// TIA Portal V17 export
// export: Created 2022-06-27T14:00:24.4169132Z, ExportSetting WithDefaults, DisplayName Totally Integrated Automation Portal, DisplayVersion V17 Update 3, DisplayName TIA Portal Openness, DisplayVersion V17 Update 3, DisplayName TIA Portal Version Control Interface, DisplayVersion V17, DisplayName SINAMICS Startdrive Advanced, DisplayVersion V17 Update1, DisplayName SINAMICS Startdrive G110M, G120, G120C, G120D, G120P, G115D, DisplayVersion V17 Update1, DisplayName SINAMICS Startdrive G130, G150, S120, S150, SINAMICS MV, S210, DisplayVersion V17 Update1, DisplayName STEP 7 Professional, DisplayVersion V17 Update 3, DisplayName STEP 7 Safety, DisplayVersion V17, DisplayName WinCC UA Professional, DisplayVersion V17 Update 3
FUNCTION_BLOCK "S0832_TRENDS_CONTROL"   // FB832, LAD
{ S7_Optimized_Access := 'TRUE' }
VERSION : 0.1
// stored: AutoNumber false, IsIECCheckEnabled false, IsRetainMemResEnabled false, MemoryReserve 100, SetENOAutomatically false, UDAEnableTagReadback false
   VAR
      ls_iIteration1 : Int;
      ls_stcConfigTrendEditC1Dry { S7_SetPoint := 'True'} : "S0831_TREND_CONFIG";
      ls_stcConfigTrendEditC1Roast { S7_SetPoint := 'True'} : "S0831_TREND_CONFIG";
      ls_stcConfigTrendEditC2Dry { S7_SetPoint := 'True'} : "S0831_TREND_CONFIG";
      ls_stcConfigTrendEditC2Roast { S7_SetPoint := 'True'} : "S0831_TREND_CONFIG";
      ls_stcConfigTrendVisuC1Dry { S7_SetPoint := 'True'} : "S0831_TREND_CONFIG";
      ls_stcConfigTrendVisuC1Roast { S7_SetPoint := 'True'} : "S0831_TREND_CONFIG";
      ls_stcConfigTrendVisuC2Dry { S7_SetPoint := 'True'} : "S0831_TREND_CONFIG";
      ls_stcConfigTrendVisuC2Roast { S7_SetPoint := 'True'} : "S0831_TREND_CONFIG";
   END_VAR
   VAR_TEMP   // added for the SCL form of the ladder/FBD networks
      _w1 : Bool;
   END_VAR
BEGIN

REGION Network 1 (SCL): SCL transferencia de valores da receita em edicao para o bloco de trend / Move valores edicao camara 1
   REGION Move valores das receitas em edicao para o bloco de trend
       REGION Move valores do secador para o bloco de trend
           FOR #ls_iIteration1 := 1 TO 10 DO
               // Statement section FOR
               #ls_stcConfigTrendEditC1Dry.i_arXBottom[#ls_iIteration1] := "S0921_ManipulacaoReceitas_DB".RecipeEdit.C1ProfileDry.arCoffeeTemperature[#ls_iIteration1];
               #ls_stcConfigTrendEditC1Dry.i_arYLeft[#ls_iIteration1] := "S0921_ManipulacaoReceitas_DB".RecipeEdit.C1ProfileDry.arInletTemperature[#ls_iIteration1];
               #ls_stcConfigTrendEditC1Dry.i_arYRight[#ls_iIteration1] := "S0921_ManipulacaoReceitas_DB".RecipeEdit.C1ProfileDry.arBlowerSpeed[#ls_iIteration1];
           END_FOR;
           #ls_stcConfigTrendEditC1Dry.i_rCorte := "S0921_ManipulacaoReceitas_DB".RecipeEdit.Recipe.rC1DryTemperature;
           #ls_stcConfigTrendEditC1Dry.i_rAromatizacao := 0.0;
       END_REGION
       REGION Move valores do torrador para o bloco de trend
           FOR #ls_iIteration1 := 1 TO 10 DO
               // Statement section FOR
               #ls_stcConfigTrendEditC1Roast.i_arXBottom[#ls_iIteration1] := "S0921_ManipulacaoReceitas_DB".RecipeEdit.C1ProfileRoast.arCoffeeTemperature[#ls_iIteration1];
               #ls_stcConfigTrendEditC1Roast.i_arYLeft[#ls_iIteration1] := "S0921_ManipulacaoReceitas_DB".RecipeEdit.C1ProfileRoast.arInletTemperature[#ls_iIteration1];
               #ls_stcConfigTrendEditC1Roast.i_arYRight[#ls_iIteration1] := "S0921_ManipulacaoReceitas_DB".RecipeEdit.C1ProfileRoast.arBlowerSpeed[#ls_iIteration1];
           END_FOR;
           #ls_stcConfigTrendEditC1Roast.i_rCorte := "S0921_ManipulacaoReceitas_DB".RecipeEdit.Recipe.rC1RoastCutTemperature;
           #ls_stcConfigTrendEditC1Roast.i_rAromatizacao := "S0921_ManipulacaoReceitas_DB".RecipeEdit.Recipe.rC1RoastQuenchTemperature;
       END_REGION
   END_REGION
END_REGION

REGION Network 2: Bloco de trend da edicao de receita / Chama blocos edicao camara 1
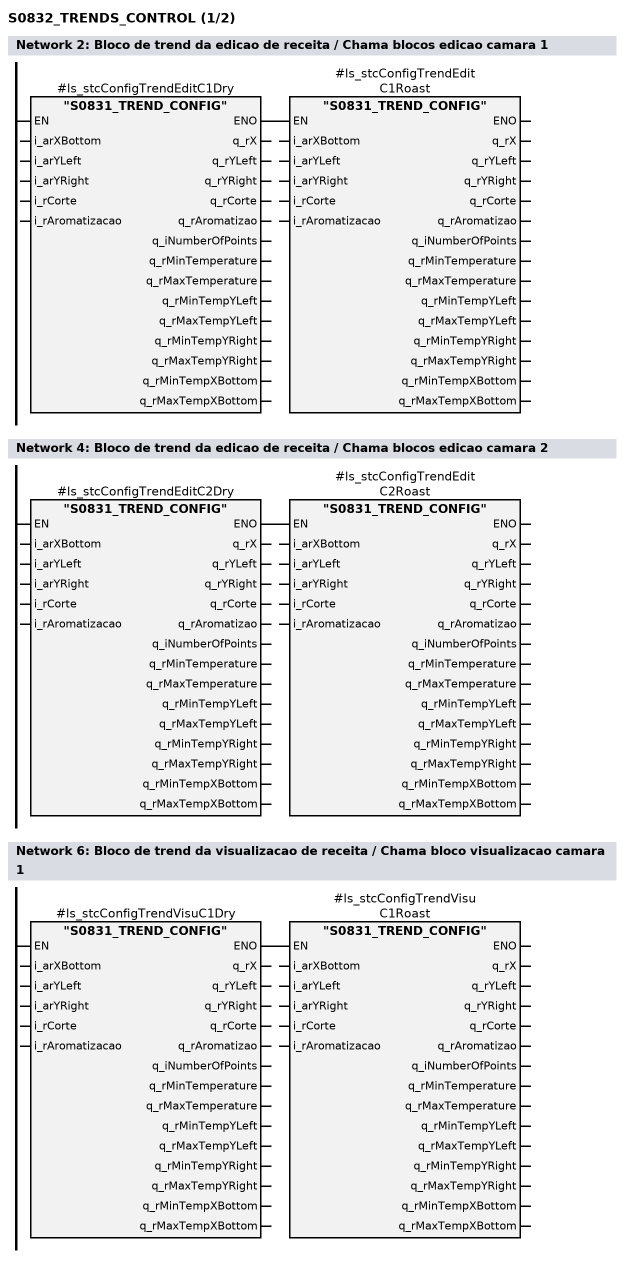
   RUNG wire#powerrail
      #ls_stcConfigTrendEditC1Dry(i_arXBottom :=, i_arYLeft :=, i_arYRight :=, i_rCorte :=, i_rAromatizacao :=, q_rX =>, q_rYLeft =>, q_rYRight =>, q_rCorte =>, q_rAromatizao =>, q_iNumberOfPoints =>, q_rMinTemperature =>, q_rMaxTemperature =>, q_rMinTempYLeft =>, q_rMaxTempYLeft =>, q_rMinTempYRight =>, q_rMaxTempYRight =>, q_rMinTempXBottom =>, q_rMaxTempXBottom =>)
      #ls_stcConfigTrendEditC1Roast(i_arXBottom :=, i_arYLeft :=, i_arYRight :=, i_rCorte :=, i_rAromatizacao :=, q_rX =>, q_rYLeft =>, q_rYRight =>, q_rCorte =>, q_rAromatizao =>, q_iNumberOfPoints =>, q_rMinTemperature =>, q_rMaxTemperature =>, q_rMinTempYLeft =>, q_rMaxTempYLeft =>, q_rMinTempYRight =>, q_rMaxTempYRight =>, q_rMinTempXBottom =>, q_rMaxTempXBottom =>)
   END_RUNG
   // the same network as SCL:
   #ls_stcConfigTrendEditC1Dry(ENO => #_w1);   // "S0831_TREND_CONFIG"
   IF #_w1 THEN
       #ls_stcConfigTrendEditC1Roast();   // "S0831_TREND_CONFIG"
   END_IF;
END_REGION

REGION Network 3 (SCL): SCL transferencia de valores da receita em edicao para o bloco de trend / Move valores edicao camara 2
   REGION Move valores das receitas em edicao para o bloco de trend
       REGION Move valores do secador para o bloco de trend
           FOR #ls_iIteration1 := 1 TO 10 DO
               // Statement section FOR
               #ls_stcConfigTrendEditC2Dry.i_arXBottom[#ls_iIteration1] := "S0921_ManipulacaoReceitas_DB".RecipeEdit.C2ProfileDry.arCoffeeTemperature[#ls_iIteration1];
               #ls_stcConfigTrendEditC2Dry.i_arYLeft[#ls_iIteration1] := "S0921_ManipulacaoReceitas_DB".RecipeEdit.C2ProfileDry.arInletTemperature[#ls_iIteration1];
               #ls_stcConfigTrendEditC2Dry.i_arYRight[#ls_iIteration1] := "S0921_ManipulacaoReceitas_DB".RecipeEdit.C2ProfileDry.arBlowerSpeed[#ls_iIteration1];
           END_FOR;
           #ls_stcConfigTrendEditC2Dry.i_rCorte := "S0921_ManipulacaoReceitas_DB".RecipeEdit.Recipe.rC2DryTemperature;
           #ls_stcConfigTrendEditC2Dry.i_rAromatizacao := 0.0;
       END_REGION
       REGION Move valores do torrador para o bloco de trend
           FOR #ls_iIteration1 := 1 TO 10 DO
               // Statement section FOR
               #ls_stcConfigTrendEditC2Roast.i_arXBottom[#ls_iIteration1] := "S0921_ManipulacaoReceitas_DB".RecipeEdit.C2ProfileRoast.arCoffeeTemperature[#ls_iIteration1];
               #ls_stcConfigTrendEditC2Roast.i_arYLeft[#ls_iIteration1] := "S0921_ManipulacaoReceitas_DB".RecipeEdit.C2ProfileRoast.arInletTemperature[#ls_iIteration1];
               #ls_stcConfigTrendEditC2Roast.i_arYRight[#ls_iIteration1] := "S0921_ManipulacaoReceitas_DB".RecipeEdit.C2ProfileRoast.arBlowerSpeed[#ls_iIteration1];
           END_FOR;
           #ls_stcConfigTrendEditC2Roast.i_rCorte := "S0921_ManipulacaoReceitas_DB".RecipeEdit.Recipe.rC2RoastCutTemperature;
           #ls_stcConfigTrendEditC2Roast.i_rAromatizacao := "S0921_ManipulacaoReceitas_DB".RecipeEdit.Recipe.rC2RoastQuenchTemperature;
       END_REGION
   END_REGION
END_REGION

REGION Network 4: Bloco de trend da edicao de receita / Chama blocos edicao camara 2
   RUNG wire#powerrail
      #ls_stcConfigTrendEditC2Dry(i_arXBottom :=, i_arYLeft :=, i_arYRight :=, i_rCorte :=, i_rAromatizacao :=, q_rX =>, q_rYLeft =>, q_rYRight =>, q_rCorte =>, q_rAromatizao =>, q_iNumberOfPoints =>, q_rMinTemperature =>, q_rMaxTemperature =>, q_rMinTempYLeft =>, q_rMaxTempYLeft =>, q_rMinTempYRight =>, q_rMaxTempYRight =>, q_rMinTempXBottom =>, q_rMaxTempXBottom =>)
      #ls_stcConfigTrendEditC2Roast(i_arXBottom :=, i_arYLeft :=, i_arYRight :=, i_rCorte :=, i_rAromatizacao :=, q_rX =>, q_rYLeft =>, q_rYRight =>, q_rCorte =>, q_rAromatizao =>, q_iNumberOfPoints =>, q_rMinTemperature =>, q_rMaxTemperature =>, q_rMinTempYLeft =>, q_rMaxTempYLeft =>, q_rMinTempYRight =>, q_rMaxTempYRight =>, q_rMinTempXBottom =>, q_rMaxTempXBottom =>)
   END_RUNG
   // the same network as SCL:
   #ls_stcConfigTrendEditC2Dry(ENO => #_w1);   // "S0831_TREND_CONFIG"
   IF #_w1 THEN
       #ls_stcConfigTrendEditC2Roast();   // "S0831_TREND_CONFIG"
   END_IF;
END_REGION

REGION Network 5 (SCL): SCL transferencia de valores da receita de visualizacao para o bloco de trend / Move valores visualizacao camara 1
   REGION Move valores das receitas em edicao para o bloco de trend
       REGION Move valores do secador para o bloco de trend

           #ls_stcConfigTrendVisuC1Dry.i_arXBottom[1] := "S0921_ManipulacaoReceitas_DB".ls_audtC1MachineProcess[2].ActualRecipe.rC1DryCoffeeTemperature1;
           #ls_stcConfigTrendVisuC1Dry.i_arXBottom[2] := "S0921_ManipulacaoReceitas_DB".ls_audtC1MachineProcess[2].ActualRecipe.rC1DryCoffeeTemperature2;
           #ls_stcConfigTrendVisuC1Dry.i_arXBottom[3] := "S0921_ManipulacaoReceitas_DB".ls_audtC1MachineProcess[2].ActualRecipe.rC1DryCoffeeTemperature3;
           #ls_stcConfigTrendVisuC1Dry.i_arXBottom[4] := "S0921_ManipulacaoReceitas_DB".ls_audtC1MachineProcess[2].ActualRecipe.rC1DryCoffeeTemperature4;
           #ls_stcConfigTrendVisuC1Dry.i_arXBottom[5] := "S0921_ManipulacaoReceitas_DB".ls_audtC1MachineProcess[2].ActualRecipe.rC1DryCoffeeTemperature5;
           #ls_stcConfigTrendVisuC1Dry.i_arXBottom[6] := "S0921_ManipulacaoReceitas_DB".ls_audtC1MachineProcess[2].ActualRecipe.rC1DryCoffeeTemperature6;
           #ls_stcConfigTrendVisuC1Dry.i_arXBottom[7] := "S0921_ManipulacaoReceitas_DB".ls_audtC1MachineProcess[2].ActualRecipe.rC1DryCoffeeTemperature7;
           #ls_stcConfigTrendVisuC1Dry.i_arXBottom[8] := "S0921_ManipulacaoReceitas_DB".ls_audtC1MachineProcess[2].ActualRecipe.rC1DryCoffeeTemperature8;
           #ls_stcConfigTrendVisuC1Dry.i_arXBottom[9] := "S0921_ManipulacaoReceitas_DB".ls_audtC1MachineProcess[2].ActualRecipe.rC1DryCoffeeTemperature9;
           #ls_stcConfigTrendVisuC1Dry.i_arXBottom[10] := "S0921_ManipulacaoReceitas_DB".ls_audtC1MachineProcess[2].ActualRecipe.rC1DryCoffeeTemperature10;
           #ls_stcConfigTrendVisuC1Dry.i_arYLeft[1] := "S0921_ManipulacaoReceitas_DB".ls_audtC1MachineProcess[2].ActualRecipe.rC1DryInletTemperature1;
           #ls_stcConfigTrendVisuC1Dry.i_arYLeft[2] := "S0921_ManipulacaoReceitas_DB".ls_audtC1MachineProcess[2].ActualRecipe.rC1DryInletTemperature2;
           #ls_stcConfigTrendVisuC1Dry.i_arYLeft[3] := "S0921_ManipulacaoReceitas_DB".ls_audtC1MachineProcess[2].ActualRecipe.rC1DryInletTemperature3;
           #ls_stcConfigTrendVisuC1Dry.i_arYLeft[4] := "S0921_ManipulacaoReceitas_DB".ls_audtC1MachineProcess[2].ActualRecipe.rC1DryInletTemperature4;
           #ls_stcConfigTrendVisuC1Dry.i_arYLeft[5] := "S0921_ManipulacaoReceitas_DB".ls_audtC1MachineProcess[2].ActualRecipe.rC1DryInletTemperature5;
           #ls_stcConfigTrendVisuC1Dry.i_arYLeft[6] := "S0921_ManipulacaoReceitas_DB".ls_audtC1MachineProcess[2].ActualRecipe.rC1DryInletTemperature6;
           #ls_stcConfigTrendVisuC1Dry.i_arYLeft[7] := "S0921_ManipulacaoReceitas_DB".ls_audtC1MachineProcess[2].ActualRecipe.rC1DryInletTemperature7;
           #ls_stcConfigTrendVisuC1Dry.i_arYLeft[8] := "S0921_ManipulacaoReceitas_DB".ls_audtC1MachineProcess[2].ActualRecipe.rC1DryInletTemperature8;
           #ls_stcConfigTrendVisuC1Dry.i_arYLeft[9] := "S0921_ManipulacaoReceitas_DB".ls_audtC1MachineProcess[2].ActualRecipe.rC1DryInletTemperature9;
           #ls_stcConfigTrendVisuC1Dry.i_arYLeft[10] := "S0921_ManipulacaoReceitas_DB".ls_audtC1MachineProcess[2].ActualRecipe.rC1DryInletTemperature10;
           #ls_stcConfigTrendVisuC1Dry.i_arYRight[1] := "S0921_ManipulacaoReceitas_DB".ls_audtC1MachineProcess[2].ActualRecipe.rC1DryBlowerSpeed1;
           #ls_stcConfigTrendVisuC1Dry.i_arYRight[2] := "S0921_ManipulacaoReceitas_DB".ls_audtC1MachineProcess[2].ActualRecipe.rC1DryBlowerSpeed2;
           #ls_stcConfigTrendVisuC1Dry.i_arYRight[3] := "S0921_ManipulacaoReceitas_DB".ls_audtC1MachineProcess[2].ActualRecipe.rC1DryBlowerSpeed3;
           #ls_stcConfigTrendVisuC1Dry.i_arYRight[4] := "S0921_ManipulacaoReceitas_DB".ls_audtC1MachineProcess[2].ActualRecipe.rC1DryBlowerSpeed4;
           #ls_stcConfigTrendVisuC1Dry.i_arYRight[5] := "S0921_ManipulacaoReceitas_DB".ls_audtC1MachineProcess[2].ActualRecipe.rC1DryBlowerSpeed5;
           #ls_stcConfigTrendVisuC1Dry.i_arYRight[6] := "S0921_ManipulacaoReceitas_DB".ls_audtC1MachineProcess[2].ActualRecipe.rC1DryBlowerSpeed6;
           #ls_stcConfigTrendVisuC1Dry.i_arYRight[7] := "S0921_ManipulacaoReceitas_DB".ls_audtC1MachineProcess[2].ActualRecipe.rC1DryBlowerSpeed7;
           #ls_stcConfigTrendVisuC1Dry.i_arYRight[8] := "S0921_ManipulacaoReceitas_DB".ls_audtC1MachineProcess[2].ActualRecipe.rC1DryBlowerSpeed8;
           #ls_stcConfigTrendVisuC1Dry.i_arYRight[9] := "S0921_ManipulacaoReceitas_DB".ls_audtC1MachineProcess[2].ActualRecipe.rC1DryBlowerSpeed9;
           #ls_stcConfigTrendVisuC1Dry.i_arYRight[10] := "S0921_ManipulacaoReceitas_DB".ls_audtC1MachineProcess[2].ActualRecipe.rC1DryBlowerSpeed10;
           #ls_stcConfigTrendVisuC1Dry.i_rCorte := "S0921_ManipulacaoReceitas_DB".ls_audtC1MachineProcess[2].ActualRecipe.rC1DryTemperature;
           #ls_stcConfigTrendVisuC1Dry.i_rAromatizacao := 0.0;

       END_REGION
       REGION Move valores do torrador para o bloco de trend

           #ls_stcConfigTrendVisuC1Roast.i_arXBottom[1] := "S0921_ManipulacaoReceitas_DB".ls_audtC1MachineProcess[2].ActualRecipe.rC1RoastCoffeeTemperature1;
           #ls_stcConfigTrendVisuC1Roast.i_arXBottom[2] := "S0921_ManipulacaoReceitas_DB".ls_audtC1MachineProcess[2].ActualRecipe.rC1RoastCoffeeTemperature2;
           #ls_stcConfigTrendVisuC1Roast.i_arXBottom[3] := "S0921_ManipulacaoReceitas_DB".ls_audtC1MachineProcess[2].ActualRecipe.rC1RoastCoffeeTemperature3;
           #ls_stcConfigTrendVisuC1Roast.i_arXBottom[4] := "S0921_ManipulacaoReceitas_DB".ls_audtC1MachineProcess[2].ActualRecipe.rC1RoastCoffeeTemperature4;
           #ls_stcConfigTrendVisuC1Roast.i_arXBottom[5] := "S0921_ManipulacaoReceitas_DB".ls_audtC1MachineProcess[2].ActualRecipe.rC1RoastCoffeeTemperature5;
           #ls_stcConfigTrendVisuC1Roast.i_arXBottom[6] := "S0921_ManipulacaoReceitas_DB".ls_audtC1MachineProcess[2].ActualRecipe.rC1RoastCoffeeTemperature6;
           #ls_stcConfigTrendVisuC1Roast.i_arXBottom[7] := "S0921_ManipulacaoReceitas_DB".ls_audtC1MachineProcess[2].ActualRecipe.rC1RoastCoffeeTemperature7;
           #ls_stcConfigTrendVisuC1Roast.i_arXBottom[8] := "S0921_ManipulacaoReceitas_DB".ls_audtC1MachineProcess[2].ActualRecipe.rC1RoastCoffeeTemperature8;
           #ls_stcConfigTrendVisuC1Roast.i_arXBottom[9] := "S0921_ManipulacaoReceitas_DB".ls_audtC1MachineProcess[2].ActualRecipe.rC1RoastCoffeeTemperature9;
           #ls_stcConfigTrendVisuC1Roast.i_arXBottom[10] := "S0921_ManipulacaoReceitas_DB".ls_audtC1MachineProcess[2].ActualRecipe.rC1RoastCoffeeTemperature10;
           #ls_stcConfigTrendVisuC1Roast.i_arYLeft[1] := "S0921_ManipulacaoReceitas_DB".ls_audtC1MachineProcess[2].ActualRecipe.rC1RoastInletTemperature1;
           #ls_stcConfigTrendVisuC1Roast.i_arYLeft[2] := "S0921_ManipulacaoReceitas_DB".ls_audtC1MachineProcess[2].ActualRecipe.rC1RoastInletTemperature2;
           #ls_stcConfigTrendVisuC1Roast.i_arYLeft[3] := "S0921_ManipulacaoReceitas_DB".ls_audtC1MachineProcess[2].ActualRecipe.rC1RoastInletTemperature3;
           #ls_stcConfigTrendVisuC1Roast.i_arYLeft[4] := "S0921_ManipulacaoReceitas_DB".ls_audtC1MachineProcess[2].ActualRecipe.rC1RoastInletTemperature4;
           #ls_stcConfigTrendVisuC1Roast.i_arYLeft[5] := "S0921_ManipulacaoReceitas_DB".ls_audtC1MachineProcess[2].ActualRecipe.rC1RoastInletTemperature5;
           #ls_stcConfigTrendVisuC1Roast.i_arYLeft[6] := "S0921_ManipulacaoReceitas_DB".ls_audtC1MachineProcess[2].ActualRecipe.rC1RoastInletTemperature6;
           #ls_stcConfigTrendVisuC1Roast.i_arYLeft[7] := "S0921_ManipulacaoReceitas_DB".ls_audtC1MachineProcess[2].ActualRecipe.rC1RoastInletTemperature7;
           #ls_stcConfigTrendVisuC1Roast.i_arYLeft[8] := "S0921_ManipulacaoReceitas_DB".ls_audtC1MachineProcess[2].ActualRecipe.rC1RoastInletTemperature8;
           #ls_stcConfigTrendVisuC1Roast.i_arYLeft[9] := "S0921_ManipulacaoReceitas_DB".ls_audtC1MachineProcess[2].ActualRecipe.rC1RoastInletTemperature9;
           #ls_stcConfigTrendVisuC1Roast.i_arYLeft[10] := "S0921_ManipulacaoReceitas_DB".ls_audtC1MachineProcess[2].ActualRecipe.rC1RoastInletTemperature10;
           #ls_stcConfigTrendVisuC1Roast.i_arYRight[1] := "S0921_ManipulacaoReceitas_DB".ls_audtC1MachineProcess[2].ActualRecipe.rC1RoastBlowerSpeed1;
           #ls_stcConfigTrendVisuC1Roast.i_arYRight[2] := "S0921_ManipulacaoReceitas_DB".ls_audtC1MachineProcess[2].ActualRecipe.rC1RoastBlowerSpeed2;
           #ls_stcConfigTrendVisuC1Roast.i_arYRight[3] := "S0921_ManipulacaoReceitas_DB".ls_audtC1MachineProcess[2].ActualRecipe.rC1RoastBlowerSpeed3;
           #ls_stcConfigTrendVisuC1Roast.i_arYRight[4] := "S0921_ManipulacaoReceitas_DB".ls_audtC1MachineProcess[2].ActualRecipe.rC1RoastBlowerSpeed4;
           #ls_stcConfigTrendVisuC1Roast.i_arYRight[5] := "S0921_ManipulacaoReceitas_DB".ls_audtC1MachineProcess[2].ActualRecipe.rC1RoastBlowerSpeed5;
           #ls_stcConfigTrendVisuC1Roast.i_arYRight[6] := "S0921_ManipulacaoReceitas_DB".ls_audtC1MachineProcess[2].ActualRecipe.rC1RoastBlowerSpeed6;
           #ls_stcConfigTrendVisuC1Roast.i_arYRight[7] := "S0921_ManipulacaoReceitas_DB".ls_audtC1MachineProcess[2].ActualRecipe.rC1RoastBlowerSpeed7;
           #ls_stcConfigTrendVisuC1Roast.i_arYRight[8] := "S0921_ManipulacaoReceitas_DB".ls_audtC1MachineProcess[2].ActualRecipe.rC1RoastBlowerSpeed8;
           #ls_stcConfigTrendVisuC1Roast.i_arYRight[9] := "S0921_ManipulacaoReceitas_DB".ls_audtC1MachineProcess[2].ActualRecipe.rC1RoastBlowerSpeed9;
           #ls_stcConfigTrendVisuC1Roast.i_arYRight[10] := "S0921_ManipulacaoReceitas_DB".ls_audtC1MachineProcess[2].ActualRecipe.rC1RoastBlowerSpeed10;
           #ls_stcConfigTrendVisuC1Roast.i_rCorte := "S0921_ManipulacaoReceitas_DB".ls_audtC1MachineProcess[2].ActualRecipe.rC1RoastCutTemperature;
           #ls_stcConfigTrendVisuC1Roast.i_rAromatizacao := "S0921_ManipulacaoReceitas_DB".ls_audtC1MachineProcess[2].ActualRecipe.rC1RoastQuenchTemperature;

       END_REGION
   END_REGION
END_REGION

REGION Network 6: Bloco de trend da visualizacao de receita / Chama bloco visualizacao camara 1
   RUNG wire#powerrail
      #ls_stcConfigTrendVisuC1Dry(i_arXBottom :=, i_arYLeft :=, i_arYRight :=, i_rCorte :=, i_rAromatizacao :=, q_rX =>, q_rYLeft =>, q_rYRight =>, q_rCorte =>, q_rAromatizao =>, q_iNumberOfPoints =>, q_rMinTemperature =>, q_rMaxTemperature =>, q_rMinTempYLeft =>, q_rMaxTempYLeft =>, q_rMinTempYRight =>, q_rMaxTempYRight =>, q_rMinTempXBottom =>, q_rMaxTempXBottom =>)
      #ls_stcConfigTrendVisuC1Roast(i_arXBottom :=, i_arYLeft :=, i_arYRight :=, i_rCorte :=, i_rAromatizacao :=, q_rX =>, q_rYLeft =>, q_rYRight =>, q_rCorte =>, q_rAromatizao =>, q_iNumberOfPoints =>, q_rMinTemperature =>, q_rMaxTemperature =>, q_rMinTempYLeft =>, q_rMaxTempYLeft =>, q_rMinTempYRight =>, q_rMaxTempYRight =>, q_rMinTempXBottom =>, q_rMaxTempXBottom =>)
   END_RUNG
   // the same network as SCL:
   #ls_stcConfigTrendVisuC1Dry(ENO => #_w1);   // "S0831_TREND_CONFIG"
   IF #_w1 THEN
       #ls_stcConfigTrendVisuC1Roast();   // "S0831_TREND_CONFIG"
   END_IF;
END_REGION

REGION Network 7 (SCL): SCL transferencia de valores da receita de visualizacao para o bloco de trend / Move valores visualizacao camara 2
   REGION Move valores das receitas em edicao para o bloco de trend
       REGION Move valores do secador para o bloco de trend

           #ls_stcConfigTrendVisuC2Dry.i_arXBottom[1] := "S0921_ManipulacaoReceitas_DB".ls_audtC2MachineProcess[2].ActualRecipe.rC2DryCoffeeTemperature1;
           #ls_stcConfigTrendVisuC2Dry.i_arXBottom[2] := "S0921_ManipulacaoReceitas_DB".ls_audtC2MachineProcess[2].ActualRecipe.rC2DryCoffeeTemperature2;
           #ls_stcConfigTrendVisuC2Dry.i_arXBottom[3] := "S0921_ManipulacaoReceitas_DB".ls_audtC2MachineProcess[2].ActualRecipe.rC2DryCoffeeTemperature3;
           #ls_stcConfigTrendVisuC2Dry.i_arXBottom[4] := "S0921_ManipulacaoReceitas_DB".ls_audtC2MachineProcess[2].ActualRecipe.rC2DryCoffeeTemperature4;
           #ls_stcConfigTrendVisuC2Dry.i_arXBottom[5] := "S0921_ManipulacaoReceitas_DB".ls_audtC2MachineProcess[2].ActualRecipe.rC2DryCoffeeTemperature5;
           #ls_stcConfigTrendVisuC2Dry.i_arXBottom[6] := "S0921_ManipulacaoReceitas_DB".ls_audtC2MachineProcess[2].ActualRecipe.rC2DryCoffeeTemperature6;
           #ls_stcConfigTrendVisuC2Dry.i_arXBottom[7] := "S0921_ManipulacaoReceitas_DB".ls_audtC2MachineProcess[2].ActualRecipe.rC2DryCoffeeTemperature7;
           #ls_stcConfigTrendVisuC2Dry.i_arXBottom[8] := "S0921_ManipulacaoReceitas_DB".ls_audtC2MachineProcess[2].ActualRecipe.rC2DryCoffeeTemperature8;
           #ls_stcConfigTrendVisuC2Dry.i_arXBottom[9] := "S0921_ManipulacaoReceitas_DB".ls_audtC2MachineProcess[2].ActualRecipe.rC2DryCoffeeTemperature9;
           #ls_stcConfigTrendVisuC2Dry.i_arXBottom[10] := "S0921_ManipulacaoReceitas_DB".ls_audtC2MachineProcess[2].ActualRecipe.rC2DryCoffeeTemperature10;
           #ls_stcConfigTrendVisuC2Dry.i_arYLeft[1] := "S0921_ManipulacaoReceitas_DB".ls_audtC2MachineProcess[2].ActualRecipe.rC2DryInletTemperature1;
           #ls_stcConfigTrendVisuC2Dry.i_arYLeft[2] := "S0921_ManipulacaoReceitas_DB".ls_audtC2MachineProcess[2].ActualRecipe.rC2DryInletTemperature2;
           #ls_stcConfigTrendVisuC2Dry.i_arYLeft[3] := "S0921_ManipulacaoReceitas_DB".ls_audtC2MachineProcess[2].ActualRecipe.rC2DryInletTemperature3;
           #ls_stcConfigTrendVisuC2Dry.i_arYLeft[4] := "S0921_ManipulacaoReceitas_DB".ls_audtC2MachineProcess[2].ActualRecipe.rC2DryInletTemperature4;
           #ls_stcConfigTrendVisuC2Dry.i_arYLeft[5] := "S0921_ManipulacaoReceitas_DB".ls_audtC2MachineProcess[2].ActualRecipe.rC2DryInletTemperature5;
           #ls_stcConfigTrendVisuC2Dry.i_arYLeft[6] := "S0921_ManipulacaoReceitas_DB".ls_audtC2MachineProcess[2].ActualRecipe.rC2DryInletTemperature6;
           #ls_stcConfigTrendVisuC2Dry.i_arYLeft[7] := "S0921_ManipulacaoReceitas_DB".ls_audtC2MachineProcess[2].ActualRecipe.rC2DryInletTemperature7;
           #ls_stcConfigTrendVisuC2Dry.i_arYLeft[8] := "S0921_ManipulacaoReceitas_DB".ls_audtC2MachineProcess[2].ActualRecipe.rC2DryInletTemperature8;
           #ls_stcConfigTrendVisuC2Dry.i_arYLeft[9] := "S0921_ManipulacaoReceitas_DB".ls_audtC2MachineProcess[2].ActualRecipe.rC2DryInletTemperature9;
           #ls_stcConfigTrendVisuC2Dry.i_arYLeft[10] := "S0921_ManipulacaoReceitas_DB".ls_audtC2MachineProcess[2].ActualRecipe.rC2DryInletTemperature10;
           #ls_stcConfigTrendVisuC2Dry.i_arYRight[1] := "S0921_ManipulacaoReceitas_DB".ls_audtC2MachineProcess[2].ActualRecipe.rC2DryBlowerSpeed1;
           #ls_stcConfigTrendVisuC2Dry.i_arYRight[2] := "S0921_ManipulacaoReceitas_DB".ls_audtC2MachineProcess[2].ActualRecipe.rC2DryBlowerSpeed2;
           #ls_stcConfigTrendVisuC2Dry.i_arYRight[3] := "S0921_ManipulacaoReceitas_DB".ls_audtC2MachineProcess[2].ActualRecipe.rC2DryBlowerSpeed3;
           #ls_stcConfigTrendVisuC2Dry.i_arYRight[4] := "S0921_ManipulacaoReceitas_DB".ls_audtC2MachineProcess[2].ActualRecipe.rC2DryBlowerSpeed4;
           #ls_stcConfigTrendVisuC2Dry.i_arYRight[5] := "S0921_ManipulacaoReceitas_DB".ls_audtC2MachineProcess[2].ActualRecipe.rC2DryBlowerSpeed5;
           #ls_stcConfigTrendVisuC2Dry.i_arYRight[6] := "S0921_ManipulacaoReceitas_DB".ls_audtC2MachineProcess[2].ActualRecipe.rC2DryBlowerSpeed6;
           #ls_stcConfigTrendVisuC2Dry.i_arYRight[7] := "S0921_ManipulacaoReceitas_DB".ls_audtC2MachineProcess[2].ActualRecipe.rC2DryBlowerSpeed7;
           #ls_stcConfigTrendVisuC2Dry.i_arYRight[8] := "S0921_ManipulacaoReceitas_DB".ls_audtC2MachineProcess[2].ActualRecipe.rC2DryBlowerSpeed8;
           #ls_stcConfigTrendVisuC2Dry.i_arYRight[9] := "S0921_ManipulacaoReceitas_DB".ls_audtC2MachineProcess[2].ActualRecipe.rC2DryBlowerSpeed9;
           #ls_stcConfigTrendVisuC2Dry.i_arYRight[10] := "S0921_ManipulacaoReceitas_DB".ls_audtC2MachineProcess[2].ActualRecipe.rC2DryBlowerSpeed10;
           #ls_stcConfigTrendVisuC2Dry.i_rCorte := "S0921_ManipulacaoReceitas_DB".ls_audtC2MachineProcess[2].ActualRecipe.rC2DryTemperature;
           #ls_stcConfigTrendVisuC2Dry.i_rAromatizacao := 0.0;

       END_REGION
       REGION Move valores do torrador para o bloco de trend

           #ls_stcConfigTrendVisuC2Roast.i_arXBottom[1] := "S0921_ManipulacaoReceitas_DB".ls_audtC2MachineProcess[2].ActualRecipe.rC2RoastCoffeeTemperature1;
           #ls_stcConfigTrendVisuC2Roast.i_arXBottom[2] := "S0921_ManipulacaoReceitas_DB".ls_audtC2MachineProcess[2].ActualRecipe.rC2RoastCoffeeTemperature2;
           #ls_stcConfigTrendVisuC2Roast.i_arXBottom[3] := "S0921_ManipulacaoReceitas_DB".ls_audtC2MachineProcess[2].ActualRecipe.rC2RoastCoffeeTemperature3;
           #ls_stcConfigTrendVisuC2Roast.i_arXBottom[4] := "S0921_ManipulacaoReceitas_DB".ls_audtC2MachineProcess[2].ActualRecipe.rC2RoastCoffeeTemperature4;
           #ls_stcConfigTrendVisuC2Roast.i_arXBottom[5] := "S0921_ManipulacaoReceitas_DB".ls_audtC2MachineProcess[2].ActualRecipe.rC2RoastCoffeeTemperature5;
           #ls_stcConfigTrendVisuC2Roast.i_arXBottom[6] := "S0921_ManipulacaoReceitas_DB".ls_audtC2MachineProcess[2].ActualRecipe.rC2RoastCoffeeTemperature6;
           #ls_stcConfigTrendVisuC2Roast.i_arXBottom[7] := "S0921_ManipulacaoReceitas_DB".ls_audtC2MachineProcess[2].ActualRecipe.rC2RoastCoffeeTemperature7;
           #ls_stcConfigTrendVisuC2Roast.i_arXBottom[8] := "S0921_ManipulacaoReceitas_DB".ls_audtC2MachineProcess[2].ActualRecipe.rC2RoastCoffeeTemperature8;
           #ls_stcConfigTrendVisuC2Roast.i_arXBottom[9] := "S0921_ManipulacaoReceitas_DB".ls_audtC2MachineProcess[2].ActualRecipe.rC2RoastCoffeeTemperature9;
           #ls_stcConfigTrendVisuC2Roast.i_arXBottom[10] := "S0921_ManipulacaoReceitas_DB".ls_audtC2MachineProcess[2].ActualRecipe.rC2RoastCoffeeTemperature10;
           #ls_stcConfigTrendVisuC2Roast.i_arYLeft[1] := "S0921_ManipulacaoReceitas_DB".ls_audtC2MachineProcess[2].ActualRecipe.rC2RoastInletTemperature1;
           #ls_stcConfigTrendVisuC2Roast.i_arYLeft[2] := "S0921_ManipulacaoReceitas_DB".ls_audtC2MachineProcess[2].ActualRecipe.rC2RoastInletTemperature2;
           #ls_stcConfigTrendVisuC2Roast.i_arYLeft[3] := "S0921_ManipulacaoReceitas_DB".ls_audtC2MachineProcess[2].ActualRecipe.rC2RoastInletTemperature3;
           #ls_stcConfigTrendVisuC2Roast.i_arYLeft[4] := "S0921_ManipulacaoReceitas_DB".ls_audtC2MachineProcess[2].ActualRecipe.rC2RoastInletTemperature4;
           #ls_stcConfigTrendVisuC2Roast.i_arYLeft[5] := "S0921_ManipulacaoReceitas_DB".ls_audtC2MachineProcess[2].ActualRecipe.rC2RoastInletTemperature5;
           #ls_stcConfigTrendVisuC2Roast.i_arYLeft[6] := "S0921_ManipulacaoReceitas_DB".ls_audtC2MachineProcess[2].ActualRecipe.rC2RoastInletTemperature6;
           #ls_stcConfigTrendVisuC2Roast.i_arYLeft[7] := "S0921_ManipulacaoReceitas_DB".ls_audtC2MachineProcess[2].ActualRecipe.rC2RoastInletTemperature7;
           #ls_stcConfigTrendVisuC2Roast.i_arYLeft[8] := "S0921_ManipulacaoReceitas_DB".ls_audtC2MachineProcess[2].ActualRecipe.rC2RoastInletTemperature8;
           #ls_stcConfigTrendVisuC2Roast.i_arYLeft[9] := "S0921_ManipulacaoReceitas_DB".ls_audtC2MachineProcess[2].ActualRecipe.rC2RoastInletTemperature9;
           #ls_stcConfigTrendVisuC2Roast.i_arYLeft[10] := "S0921_ManipulacaoReceitas_DB".ls_audtC2MachineProcess[2].ActualRecipe.rC2RoastInletTemperature10;
           #ls_stcConfigTrendVisuC2Roast.i_arYRight[1] := "S0921_ManipulacaoReceitas_DB".ls_audtC2MachineProcess[2].ActualRecipe.rC2RoastBlowerSpeed1;
           #ls_stcConfigTrendVisuC2Roast.i_arYRight[2] := "S0921_ManipulacaoReceitas_DB".ls_audtC2MachineProcess[2].ActualRecipe.rC2RoastBlowerSpeed2;
           #ls_stcConfigTrendVisuC2Roast.i_arYRight[3] := "S0921_ManipulacaoReceitas_DB".ls_audtC2MachineProcess[2].ActualRecipe.rC2RoastBlowerSpeed3;
           #ls_stcConfigTrendVisuC2Roast.i_arYRight[4] := "S0921_ManipulacaoReceitas_DB".ls_audtC2MachineProcess[2].ActualRecipe.rC2RoastBlowerSpeed4;
           #ls_stcConfigTrendVisuC2Roast.i_arYRight[5] := "S0921_ManipulacaoReceitas_DB".ls_audtC2MachineProcess[2].ActualRecipe.rC2RoastBlowerSpeed5;
           #ls_stcConfigTrendVisuC2Roast.i_arYRight[6] := "S0921_ManipulacaoReceitas_DB".ls_audtC2MachineProcess[2].ActualRecipe.rC2RoastBlowerSpeed6;
           #ls_stcConfigTrendVisuC2Roast.i_arYRight[7] := "S0921_ManipulacaoReceitas_DB".ls_audtC2MachineProcess[2].ActualRecipe.rC2RoastBlowerSpeed7;
           #ls_stcConfigTrendVisuC2Roast.i_arYRight[8] := "S0921_ManipulacaoReceitas_DB".ls_audtC2MachineProcess[2].ActualRecipe.rC2RoastBlowerSpeed8;
           #ls_stcConfigTrendVisuC2Roast.i_arYRight[9] := "S0921_ManipulacaoReceitas_DB".ls_audtC2MachineProcess[2].ActualRecipe.rC2RoastBlowerSpeed9;
           #ls_stcConfigTrendVisuC2Roast.i_arYRight[10] := "S0921_ManipulacaoReceitas_DB".ls_audtC2MachineProcess[2].ActualRecipe.rC2RoastBlowerSpeed10;
           #ls_stcConfigTrendVisuC2Roast.i_rCorte := "S0921_ManipulacaoReceitas_DB".ls_audtC2MachineProcess[2].ActualRecipe.rC2RoastCutTemperature;
           #ls_stcConfigTrendVisuC2Roast.i_rAromatizacao := "S0921_ManipulacaoReceitas_DB".ls_audtC2MachineProcess[2].ActualRecipe.rC2RoastQuenchTemperature;

       END_REGION
   END_REGION
END_REGION

REGION Network 8: Bloco de trend da visualizacao de receita / Chama bloco visualizacao camara 2
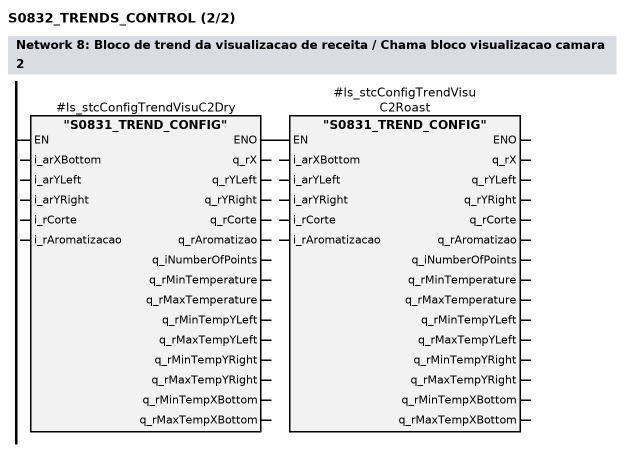
   RUNG wire#powerrail
      #ls_stcConfigTrendVisuC2Dry(i_arXBottom :=, i_arYLeft :=, i_arYRight :=, i_rCorte :=, i_rAromatizacao :=, q_rX =>, q_rYLeft =>, q_rYRight =>, q_rCorte =>, q_rAromatizao =>, q_iNumberOfPoints =>, q_rMinTemperature =>, q_rMaxTemperature =>, q_rMinTempYLeft =>, q_rMaxTempYLeft =>, q_rMinTempYRight =>, q_rMaxTempYRight =>, q_rMinTempXBottom =>, q_rMaxTempXBottom =>)
      #ls_stcConfigTrendVisuC2Roast(i_arXBottom :=, i_arYLeft :=, i_arYRight :=, i_rCorte :=, i_rAromatizacao :=, q_rX =>, q_rYLeft =>, q_rYRight =>, q_rCorte =>, q_rAromatizao =>, q_iNumberOfPoints =>, q_rMinTemperature =>, q_rMaxTemperature =>, q_rMinTempYLeft =>, q_rMaxTempYLeft =>, q_rMinTempYRight =>, q_rMaxTempYRight =>, q_rMinTempXBottom =>, q_rMaxTempXBottom =>)
   END_RUNG
   // the same network as SCL:
   #ls_stcConfigTrendVisuC2Dry(ENO => #_w1);   // "S0831_TREND_CONFIG"
   IF #_w1 THEN
       #ls_stcConfigTrendVisuC2Roast();   // "S0831_TREND_CONFIG"
   END_IF;
END_REGION
END_FUNCTION_BLOCK
